INTERFACE ITFNoodStop

END_INTERFACE

(* stored: Version 1.1.0.1
   Itf ITFNoodStop: Id {2c1ec3b4-449e-49d5-a307-daafec2f6710} *)
